{attribute 'linkalways'} 
{attribute 'no_explicit_call' := 'This FB is a CLASS and must be accessed using methods or properties'}
{attribute 'enable_dynamic_creation'}
FUNCTION_BLOCK ABSTRACT DatatypeBase EXTENDS Disposable IMPLEMENTS I_Datatype
VAR
END_VAR

METHOD PUBLIC Accept
VAR_INPUT
	Visitor : I_DatatypeVisitor;
END_VAR
Visitor.VisitDatatype(this^);
END_METHOD

PROPERTY PUBLIC ABSTRACT Address : PVOID
GET
END_GET
END_PROPERTY

METHOD PUBLIC ABSTRACT ClearReference
VAR_INPUT
END_VAR
END_METHOD

METHOD PUBLIC ABSTRACT Clone : I_Datatype
END_METHOD

PROPERTY PUBLIC ABSTRACT Datatype : T_MAXSTRING
GET
END_GET
END_PROPERTY

METHOD PROTECTED OnSerializeTypeWith
VAR_INPUT
	Serializer : I_Serializer;
END_VAR
Serializer.AddKeyString('datatype',Datatype);
END_METHOD

METHOD PUBLIC SerializeTypeWith
VAR_INPUT
	Serializer : I_Serializer;
END_VAR
Serializer.StartObject();
OnSerializeTypeWith(Serializer);
Serializer.EndObject();
END_METHOD

METHOD PUBLIC ABSTRACT SerializeWith
VAR_INPUT
	Serializer : I_Serializer;
END_VAR
END_METHOD

PROPERTY PUBLIC ABSTRACT Size : UDINT
GET
END_GET
END_PROPERTY

METHOD PUBLIC TryCopy : BOOL
VAR_INPUT
	Source : I_Datatype;
END_VAR
IF Source.Datatype <> Datatype THEN
	RETURN;
END_IF

memcpy(Address, Source.Address, Size);
END_METHOD

METHOD PUBLIC ABSTRACT TryDeserializeFrom : BOOL
VAR_INPUT
	Deserializer : I_Deserializer;
	Feedback : I_DeserializerFeedback;
END_VAR
END_METHOD

METHOD PUBLIC ABSTRACT TryMakeReferenceTo : BOOL
VAR_INPUT
	Target : I_Datatype;
END_VAR
END_METHOD

METHOD PUBLIC TryResolveAsAliasType : BOOL
VAR_INPUT
	Destination : REFERENCE TO I_AliasDatatype;
END_VAR
TryResolveAsAliasType := FALSE;
END_METHOD

METHOD PUBLIC TryResolveAsEnumType : BOOL
VAR_INPUT
	Destination : REFERENCE TO I_EnumDatatype;
END_VAR
TryResolveAsEnumType := FALSE;
END_METHOD

METHOD PUBLIC TryResolveAsStructuredType : BOOL
VAR_INPUT
	Destination : REFERENCE TO I_StructuredDatatype;
END_VAR
TryResolveAsStructuredType := FALSE;
END_METHOD

END_FUNCTION_BLOCK

(* stored: Version 1.1.0.1, ProductVersion 3.1.4024.12
   POU DatatypeBase: Id {caf70741-0fda-4312-8507-6bdd6e0bf45b}, SpecialFunc None
   Folder Protected: Id {6a05f5d0-e949-0c1c-2ebf-f6a37260ee33}
   Method Accept: Id {dd871bbb-4ec4-0283-1fd2-71cc24047cd6}
   Property Address: Id {d51246f1-c326-4bd3-ad2b-6abdbcc9c6a3}
   Get Get: Id {75c65319-5779-49e1-ac09-d48067a51f26}
   Method ClearReference: Id {4259927f-6f52-00ed-02eb-e8cf594481d2}
   Method Clone: Id {7af27274-3902-4c83-b5c8-4b63225091df}
   Property Datatype: Id {4e6b709c-3c41-0f61-1dc2-0d8936572b7d}
   Get Get: Id {0619a35f-75ef-01ba-106d-74a7e27a44d7}
   Method OnSerializeTypeWith: Id {969b142b-0816-0c8c-3581-697926ecbe26}
   Method SerializeTypeWith: Id {d792640c-a39f-4b1c-9df5-bece16fc714d}
   Method SerializeWith: Id {52279ac4-78de-4c93-a829-75eb4e6edb6e}
   Property Size: Id {d5f34be1-cf1e-4cd3-abd8-f6af95068bbf}
   Get Get: Id {fecee7eb-1948-431d-976e-3ca35711d21b}
   Method TryCopy: Id {ff5a7101-aefc-4015-bfe6-0f0bdfd3b844}
   Method TryDeserializeFrom: Id {eeb476e5-73e9-46e1-b773-fda92a913dc4}
   Method TryMakeReferenceTo: Id {aed9eb80-ebc5-03fc-0ecc-e5fedc065442}
   Method TryResolveAsAliasType: Id {55ca9292-ffda-0855-259b-60ba4748a149}
   Method TryResolveAsEnumType: Id {788e06a8-2cbf-0aa6-002d-57c7be26c3d7}
   Method TryResolveAsStructuredType: Id {ec909d59-647a-0183-1246-435cce0f434c} *)
